Yaskawa INFORM job: R1_ROBOTCALIB_WIDE.JBI

/JOB
//NAME R1_ROBOTCALIB_WIDE
///FOLDERNAME INNE
//POS
///NPOS 8,8,0,0,0,0
///TOOL 0
///POSTYPE PULSE
///PULSE
C00000=-27876,-43237,-7229,-75376,63305,45633
C00001=-27876,-43237,-7229,-75376,63305,45633
C00002=-27876,-43237,-7229,-75376,63305,45633
C00003=-27876,-43237,-7229,-75376,63305,45633
C00004=-27876,-43237,-7229,-75376,63305,45633
C00005=-176070,-22935,-50277,47271,56747,-21463
C00006=-176070,-22935,-50277,47271,56747,-21463
C00007=-27876,-43237,-7229,-75376,63305,45633
BC00000=397782,129,502200
BC00001=30680,129,502200
BC00002=2221,129,1074942
BC00003=398102,129,1074942
BC00004=397782,1152201,502200
BC00005=72685,1083409,266561
BC00006=72685,1083409,1071099
BC00007=398102,1152201,1074942
//INST
///DATE 2023/10/17 12:51
///ATTR SC,RW
///GROUP1 RB1,BS1
NOP
'COMMENT
MOVJ C00000 BC00000 VJ=0.78 PL=0
MOVJ C00001 BC00001 VJ=0.78 PL=0
MOVJ C00002 BC00002 VJ=0.78 PL=0
MOVJ C00003 BC00003 VJ=0.78 PL=0
'COMMENT
MOVJ C00004 BC00004 VJ=0.78 PL=0
MOVJ C00005 BC00005 VJ=0.78 PL=0
MOVJ C00006 BC00006 VJ=0.78 PL=0
MOVJ C00007 BC00007 VJ=0.78 PL=0
END
